(* IEC 61131-3 sources: Word/plc-course/08-counters/labs/solutions, 3 files *)

(* ---- 08-1-bottle-packing.st ---- *)
(* Lab 08-1: Bottle packing - count bottles into a box, index the full box, start again.
   Module 08 (Counters). REFERENCE SOLUTION - try the lab yourself first.

   Idea: one CTU counts bottles and its Q says "box full". A TP turns that
   moment into a box-conveyor run of exactly IndexTime. While the TP runs,
   the counter's R input is held TRUE, so the count restarts from zero and
   anything the photo-eye sees during the index is ignored.

   Another correct design keeps the count at BoxSize during the index and
   resets it when the index ends. The lab allows either. *)

PROGRAM BottlePacking
  VAR (* I/O - addresses follow the OpenPLC convention *)
    BottlePE   AT %IX0.0 : BOOL;  (* Photo-eye at the end of the infeed: TRUE while a bottle blocks the beam *)
    ResetPB    AT %IX0.1 : BOOL;  (* Count reset push-button, NO: the operator has fitted a new, empty box *)
    InfeedConv AT %QX0.0 : BOOL;  (* Infeed conveyor motor: carries bottles into the box *)
    BoxConv    AT %QX0.1 : BOOL;  (* Box conveyor motor: moves the full box out and an empty one in *)
  END_VAR
  VAR (* HMI settings and displays - part of the lab interface *)
    BoxSize     : INT := 12;      (* bottles per box, 1..48 *)
    IndexTime   : TIME := T#2s;   (* how long the box conveyor runs to index one box *)
    BottleCount : INT;            (* bottles counted into the box being filled *)
  END_VAR
  VAR RETAIN (* a production total: on a real PLC it must survive a power cut *)
    BoxesPacked : DINT;           (* full boxes; ResetPB does not touch it *)
  END_VAR
  VAR (* internal *)
    BottleCtr  : CTU;             (* counts bottles into the current box *)
    IndexPulse : TP;              (* runs the box conveyor for IndexTime *)
    BoxFull    : R_TRIG;          (* TRUE for one scan when a box becomes full *)
    CtrPV      : INT;             (* BoxSize, kept inside 1..48 *)
  END_VAR

  (* A preset of 0 or less would make the counter "full" with no bottles at
     all, and the box conveyor would index for ever. Guard the HMI value. *)
  CtrPV := LIMIT(1, BoxSize, 48);

  (* 1. Count bottles. CTU counts RISING edges of CU, so a bottle that stops
        in the beam is still one bottle. R wins over CU: while the operator
        holds Reset, or while the box is indexing, the count is held at zero
        and the counter's internal edge memory still follows the photo-eye.
        So a bottle that is in the beam when R is released is NOT counted
        again. (IndexPulse.Q is last scan's value here: the reset starts one
        scan after the box becomes full.) *)
  BottleCtr(CU := BottlePE, R := ResetPB OR IndexPulse.Q, PV := CtrPV);
  BottleCount := BottleCtr.CV;

  (* 2. Box full. Q is TRUE from the scan the count reaches the preset. It
        drops again on the next scan, when R clears the count, but a TP only
        needs a rising edge on IN: it then runs for exactly PT. *)
  IndexPulse(IN := BottleCtr.Q, PT := IndexTime);
  BoxConv := IndexPulse.Q;

  (* 3. Production total: one per full box, on the rising edge of "full". *)
  BoxFull(CLK := BottleCtr.Q);
  IF BoxFull.Q THEN
    BoxesPacked := BoxesPacked + 1;
  END_IF;

  (* 4. The infeed stops in the same scan as the last bottle is counted, stays
        stopped while the box indexes, and stops while the operator resets the
        count so that no bottle can drop into the box uncounted. *)
  InfeedConv := NOT (BottleCtr.Q OR IndexPulse.Q OR ResetPB);
END_PROGRAM

CONFIGURATION Config0
  RESOURCE Res0 ON PLC
    TASK MainTask(INTERVAL := T#10ms, PRIORITY := 0);
    PROGRAM Inst0 WITH MainTask : BottlePacking;
  END_RESOURCE
END_CONFIGURATION

(* ---- 08-2-car-park.st ---- *)
(* Lab 08-2: Car park up/down counter with capacity, FULL sign and manual preset.
   Module 08 (Counters). REFERENCE SOLUTION - try the lab yourself first.

   Why not a CTUD with PV := Capacity? It is the obvious block, but:
   - the standard leaves the counting limits to the implementation. The
     MATIEC library behind OpenPLC and plctest stops counting UP at PV, so
     cars that ignore the FULL sign would be lost from the count. Siemens
     counts on, but also counts DOWN below 0.
   - on every platform, LD loads PV, so LD could only load Capacity, not
     the attendant's count.
   So this solution counts with ADD/SUB and sets its own limits explicitly:
   never below 0, never past the INT maximum. README section 6.3 shows a
   CTUD version that works around both problems. *)

PROGRAM CarPark
  VAR (* I/O - addresses follow the OpenPLC convention *)
    EntryLoop AT %IX0.0 : BOOL;  (* Vehicle detector, entry lane: TRUE while a car is over the loop *)
    ExitLoop  AT %IX0.1 : BOOL;  (* Vehicle detector, exit lane: TRUE while a car is over the loop *)
    PresetPB  AT %IX0.2 : BOOL;  (* Attendant's preset push-button, NO: load PresetValue into the count *)
    FullSign  AT %QX0.0 : BOOL;  (* "FULL" sign at the entrance *)
  END_VAR
  VAR (* HMI settings and displays - part of the lab interface *)
    Capacity    : INT := 50;     (* number of parking spaces *)
    PresetValue : INT;           (* cars the attendant counted by walking round *)
    SpacesFree  : INT;           (* for the "spaces" sign: never negative *)
  END_VAR
  VAR RETAIN (* the cars do not leave when the power fails *)
    CarCount    : INT;           (* cars in the car park *)
  END_VAR
  VAR (* internal *)
    CarIn  : R_TRIG;             (* a car has just arrived on the entry loop *)
    CarOut : R_TRIG;             (* a car has just arrived on the exit loop *)
  END_VAR

  (* 1. Edge detection on every scan, outside any IF, so the edge memories
        always follow the loops - also while the preset button is held. *)
  CarIn(CLK := EntryLoop);
  CarOut(CLK := ExitLoop);

  (* 2. Preset has priority, like LD on a CTUD: while it is held the count
        is PresetValue (a negative entry is treated as 0) and no cars are
        counted. A car that is on a loop when the button is released has
        already been seen by the edge detector, so it is not counted late. *)
  IF PresetPB THEN
    CarCount := MAX(PresetValue, 0);
  ELSE
    (* Two separate IFs, not IF...ELSIF: a car can enter and another leave
       in the same scan, and both must be counted. *)
    IF CarIn.Q AND CarCount < 32767 THEN      (* INT limit: never wrap to -32768 *)
      CarCount := CarCount + 1;
    END_IF;
    IF CarOut.Q AND CarCount > 0 THEN         (* never below 0 *)
      CarCount := CarCount - 1;
    END_IF;
  END_IF;

  (* 3. Signs. The count may be above Capacity (drivers ignore the sign,
        motorcycles share a space ...): the FULL sign then stays on, and the
        spaces sign shows 0, not a negative number. *)
  FullSign := CarCount >= Capacity;
  SpacesFree := MAX(Capacity - CarCount, 0);
END_PROGRAM

CONFIGURATION Config0
  RESOURCE Res0 ON PLC
    TASK MainTask(INTERVAL := T#10ms, PRIORITY := 0);
    PROGRAM Inst0 WITH MainTask : CarPark;
  END_RESOURCE
END_CONFIGURATION

(* ---- 08-3-production-counts.st ---- *)
(* Lab 08-3: Production counts - good/reject counters, total, yield, shift reset.
   Module 08 (Counters). REFERENCE SOLUTION - try the lab yourself first.

   The counts are kept with ADD (Count := Count + 1 on an edge) rather than
   with CTU blocks. A CTU's reset input wins over its count input, so a pack
   that arrives in the very scan of the shift reset would be lost. Here the
   shift change is handled first and the counting afterwards, so no pack is
   ever lost. There is no preset to reach, so a CTU would add nothing. *)

PROGRAM ProductionCounts
  VAR (* I/O - addresses follow the OpenPLC convention *)
    GoodPE       AT %IX0.0 : BOOL;  (* Photo-eye on the outfeed: TRUE while an accepted pack is in the beam *)
    RejectPE     AT %IX0.1 : BOOL;  (* Photo-eye on the reject chute: TRUE while a rejected pack passes *)
    ShiftResetPB AT %IX0.2 : BOOL;  (* Shift-change push-button, NO *)
    LowYieldLamp AT %QX0.0 : BOOL;  (* Low-yield warning lamp on the line *)
  END_VAR
  VAR (* HMI settings - part of the lab interface *)
    MinSample  : DINT := 20;        (* no yield warning until this many packs this shift *)
    YieldLimit : REAL := 95.0;      (* warn when the yield is below this, % *)
  END_VAR
  VAR RETAIN (* HMI displays that must survive a power cut *)
    GoodCount       : DINT;         (* accepted packs this shift *)
    RejectCount     : DINT;         (* rejected packs this shift *)
    LastShiftGood   : DINT;         (* snapshot taken at the last shift change *)
    LastShiftReject : DINT;
    LastShiftYield  : REAL;
    LifetimeTotal   : DINT;         (* every pack since commissioning: no reset *)
  END_VAR
  VAR (* HMI displays, recalculated every scan *)
    TotalCount : DINT;              (* GoodCount + RejectCount *)
    YieldPct   : REAL;              (* 100 x good / total; 0.0 while the total is 0 *)
  END_VAR
  VAR CONSTANT
    DINT_MAX : DINT := 2147483647;  (* largest DINT: 2^31 - 1 *)
  END_VAR
  VAR (* internal *)
    GoodIn    : R_TRIG;             (* an accepted pack has just arrived *)
    RejectIn  : R_TRIG;             (* a rejected pack has just arrived *)
    ShiftEdge : R_TRIG;             (* the shift button has just been pressed *)
  END_VAR

  (* 1. Edge detection, every scan. *)
  GoodIn(CLK := GoodPE);
  RejectIn(CLK := RejectPE);
  ShiftEdge(CLK := ShiftResetPB);

  (* 2. Shift change, on the PRESS of the button only. Holding the button
        must not repeat it, or the next scan would copy the fresh zeros over
        the snapshot. Snapshot first, then clear. YieldPct still holds the
        value calculated at the end of the previous scan from these same
        counts, so it is the finished shift's yield. *)
  IF ShiftEdge.Q THEN
    LastShiftGood := GoodCount;
    LastShiftReject := RejectCount;
    LastShiftYield := YieldPct;
    GoodCount := 0;
    RejectCount := 0;
  END_IF;

  (* 3. Counting, after the shift change, so a pack arriving in the same scan
        as the reset counts in the new shift. Independent IFs: a good pack
        and a reject can arrive in the same scan. *)
  IF GoodIn.Q THEN
    GoodCount := GoodCount + 1;
  END_IF;
  IF RejectIn.Q THEN
    RejectCount := RejectCount + 1;
  END_IF;

  (* The lifetime total must never wrap round to a negative number: it stops
     at the largest DINT. (At 10 packs a second that takes about 6.8 years.) *)
  IF GoodIn.Q AND LifetimeTotal < DINT_MAX THEN
    LifetimeTotal := LifetimeTotal + 1;
  END_IF;
  IF RejectIn.Q AND LifetimeTotal < DINT_MAX THEN
    LifetimeTotal := LifetimeTotal + 1;
  END_IF;

  (* 4. Total and yield. Convert to REAL BEFORE dividing: in integer maths
        2 / 3 = 0. And never divide by zero: at power-up and just after a
        shift change the total is 0. *)
  TotalCount := GoodCount + RejectCount;
  IF TotalCount > 0 THEN
    YieldPct := 100.0 * DINT_TO_REAL(GoodCount) / DINT_TO_REAL(TotalCount);
  ELSE
    YieldPct := 0.0;
  END_IF;

  (* 5. A yield worked out from a handful of packs means little (one reject
        in the first pack of the shift is "0 %"), so only warn once the
        sample is big enough. *)
  LowYieldLamp := (TotalCount >= MinSample) AND (YieldPct < YieldLimit);
END_PROGRAM

CONFIGURATION Config0
  RESOURCE Res0 ON PLC
    TASK MainTask(INTERVAL := T#10ms, PRIORITY := 0);
    PROGRAM Inst0 WITH MainTask : ProductionCounts;
  END_RESOURCE
END_CONFIGURATION
